Universal Robots PolyScope program: circle motion edge detect.urp

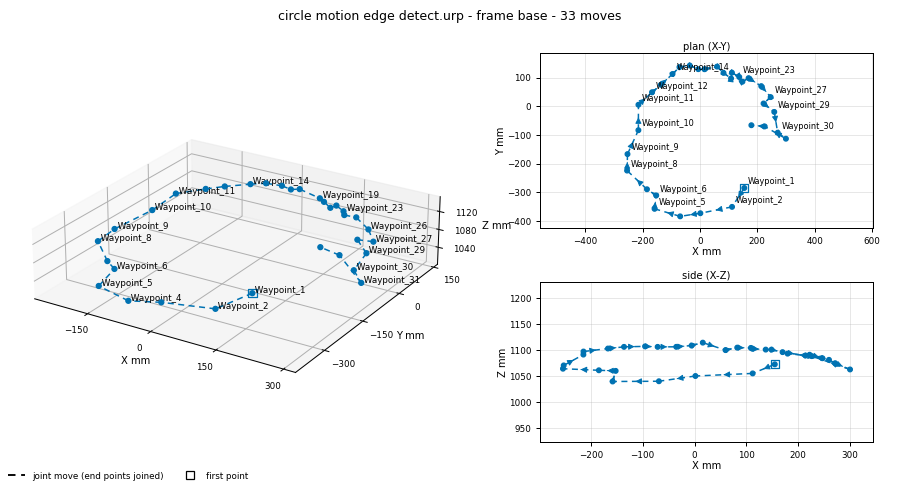
[picture p0: tool path of circle motion edge detect.urp in frame base, 33 of 33 moves have a stored position in this frame; points joined in program order, loops and branches not executed]
Program circle motion edge detect (installation=default directory=/programs/usbdisk createdIn=5.3.0.64176 lastSavedIn=5.3.0.64176 robotSerialNumber=20195500242)
Calibrated DH parameters: a=[-0.00003, -0.418785, -0.364045, -0.000016, 0.000085, 0]; d=[0.162521, -27.105222, -29.89969, 57.138732, 0.099744, 0.099563]; alpha=[1.571361, -0.002704, -0.002569, 1.570134, -1.569255, 0]; deltaTheta=[0, 0.173233, 6.492369, -0.382427, -0.000002, 0]
Robot Program (runOnlyOnce=false)
  MoveJ speed 60 deg/s, acceleration 80 deg/s^2 (useActiveTCP=true) feature=Base
    Waypoint Waypoint_1: TCP in base x=154.914 y=-284.469 z=1072.951 mm, rx=0.2997 ry=-0.5241 rz=-2.3512 rad; joints [-37.372, -111.15, 6.695, -138.52, -90.992, 169.489] deg
    Wait Sleep waitTime=2
    Waypoint Waypoint_2: TCP in base x=112.222 y=-350.291 z=1055.38 mm, rx=0.2716 ry=-0.6364 rz=-2.5729 rad; joints [-51.18, -115.112, 6.722, -132.303, -90.965, 169.471] deg; TCP offset x=0 y=0 z=0 mm, rx=0 ry=0 rz=0 rad
    Wait Sleep waitTime=2
    Waypoint Waypoint_3: TCP in base x=1.771 y=-372.471 z=1050.371 mm, rx=0.1105 ry=-0.864 rz=-2.8765 rad; joints [-70.07, -116.408, 6.715, -126.913, -94.954, 169.472] deg; TCP offset x=0 y=0 z=0 mm, rx=0 ry=0 rz=0 rad
    Wait Sleep waitTime=2
    Waypoint Waypoint_4: TCP in base x=-68.656 y=-383.358 z=1040.258 mm, rx=-0.0416 ry=0.9721 rz=2.9298 rad; joints [-81.366, -118.375, 6.714, -121.793, -94.913, 169.475] deg
    Wait Sleep waitTime=2
    Waypoint Waypoint_5: TCP in base x=-158.009 y=-357.106 z=1039.79 mm, rx=0.0714 ry=0.905 rz=2.7108 rad; joints [-95.142, -118.447, 6.717, -121.809, -94.948, 169.471] deg; TCP offset x=0 y=0 z=0 mm, rx=0 ry=0 rz=0 rad
    Wait Sleep waitTime=2
    Waypoint Waypoint_6: TCP in base x=-152.118 y=-310.493 z=1060.277 mm, rx=0.1283 ry=0.8737 rz=2.7 rad; joints [-95.524, -114.683, 6.715, -126.752, -97.143, 169.442] deg
    Wait Sleep waitTime=2
    Waypoint Waypoint_7: TCP in base x=-184.474 y=-288.892 z=1061.417 mm, rx=0.1713 ry=0.8461 rz=2.5969 rad; joints [-101.799, -114.48, 6.716, -126.753, -97.157, 169.441] deg
    Wait Sleep waitTime=2
    Waypoint Waypoint_8: TCP in base x=-253.787 y=-223.74 z=1064.438 mm, rx=0.2688 ry=0.6858 rz=2.3492 rad; joints [-117.741, -113.528, 6.714, -131.132, -97.725, 169.066] deg
    Wait Sleep waitTime=2
    Waypoint Waypoint_9: TCP in base x=-252.359 y=-166.285 z=1070.795 mm, rx=0.4935 ry=0.5953 rz=1.8556 rad; joints [-127.845, -111.078, 6.717, -133.526, -111.538, 154.842] deg
    Wait Sleep waitTime=2
    Waypoint Waypoint_10: TCP in base x=-214.374 y=-83.001 z=1091.69 mm, rx=0.5264 ry=0.6522 rz=1.7224 rad; joints [-133.832, -106.245, 6.744, -133.513, -111.607, 154.823] deg
    Wait Sleep waitTime=2
    Waypoint Waypoint_11: TCP in base x=-214.184 y=5.835 z=1097.569 mm, rx=0.5409 ry=0.5799 rz=1.432 rad; joints [-152.715, -105.043, 6.723, -133.525, -107.815, 154.808] deg
    Wait Sleep waitTime=2
    Waypoint Waypoint_12: TCP in base x=-166.957 y=49.058 z=1103.38 mm, rx=0.5833 ry=0.3942 rz=1.2936 rad; joints [-161.963, -100.794, 6.708, -143.941, -110.807, 154.793] deg
    Wait Sleep waitTime=2
    Waypoint Waypoint_13: TCP in base x=-136 y=75.302 z=1106.619 mm, rx=0.5655 ry=0.4183 rz=0.9843 rad; joints [-169.727, -99.399, 6.733, -143.942, -110.805, 144.497] deg
    Wait Sleep waitTime=2
    Waypoint Waypoint_14: TCP in base x=-95.348 y=112.97 z=1107.58 mm, rx=0.7237 ry=0.4441 rz=0.5929 rad; joints [-189.526, -100.482, 6.716, -132.699, -112.568, 144.513] deg
    Wait Sleep waitTime=2
    Waypoint Waypoint_15: TCP in base x=-71.129 y=136.814 z=1106.589 mm, rx=0.7608 ry=0.3382 rz=0.3554 rad; joints [-204.168, -100.977, 6.716, -132.715, -112.525, 144.514] deg; TCP offset x=0 y=0 z=0 mm, rx=0 ry=0 rz=0 rad
    Wait Sleep waitTime=2
    Waypoint Waypoint_16: TCP in base x=-35.171 y=142.592 z=1106.68 mm, rx=0.6766 ry=0.1374 rz=0.2072 rad; joints [-215.551, -98.736, 6.732, -144.572, -112.524, 144.514] deg; TCP offset x=0 y=0 z=0 mm, rx=0 ry=0 rz=0 rad
    Wait Sleep waitTime=2
    Waypoint Waypoint_17: TCP in base x=-5.632 y=129.883 z=1109.151 mm, rx=0.6981 ry=0.1269 rz=0.1239 rad; joints [-220.201, -97.319, 6.732, -144.572, -112.523, 144.518] deg; TCP offset x=0 y=0 z=0 mm, rx=0 ry=0 rz=0 rad
    Wait Sleep waitTime=2
    Waypoint Waypoint_18: TCP in base x=15.993 y=129.668 z=1114.734 mm, rx=0.6763 ry=0.2381 rz=0.2822 rad; joints [-220.316, -97.009, 6.71, -140.826, -104.269, 152.017] deg; TCP offset x=0 y=0 z=0 mm, rx=0 ry=0 rz=0 rad
    Wait Sleep waitTime=2
    Waypoint Waypoint_19: TCP in base x=59.885 y=138.766 z=1100.329 mm, rx=0.6524 ry=-0.0476 rz=0.1475 rad; joints [-246.927, -85.881, -20.149, -128.724, -103.816, 169.846] deg; TCP offset x=0 y=0 z=0 mm, rx=0 ry=0 rz=0 rad
    Wait Sleep waitTime=2
    Waypoint Waypoint_20: TCP in base x=82.45 y=116.928 z=1105.125 mm, rx=0.6534 ry=0.2343 rz=-0.2354 rad; joints [-246.975, -84.634, -20.096, -125.99, -96.737, 145.064] deg; TCP offset x=0 y=0 z=0 mm, rx=0 ry=0 rz=0 rad
    Wait Sleep waitTime=2
    Waypoint Waypoint_21: TCP in base x=108.815 y=97.49 z=1104.594 mm, rx=0.6598 ry=0.1537 rz=-0.5229 rad; joints [-261.813, -84.817, -20.066, -127.18, -96.744, 142.73] deg; TCP offset x=0 y=0 z=0 mm, rx=0 ry=0 rz=0 rad
    Wait Sleep waitTime=2
    Waypoint Waypoint_22: TCP in base x=111.731 y=117.75 z=1102.96 mm, rx=0.6639 ry=0.218 rz=-0.5839 rad; joints [-262.695, -86.632, -20.04, -123.996, -94.334, 139.125] deg
    Wait Sleep waitTime=2
    Waypoint Waypoint_23: TCP in base x=137.4 y=102.53 z=1101.341 mm, rx=0.7665 ry=0.2773 rz=-0.7011 rad; joints [-271.96, -88.103, -20.048, -116.073, -89.774, 139.116] deg
    Wait Sleep waitTime=2
    Waypoint Waypoint_24: TCP in base x=148.462 y=86.299 z=1101.282 mm, rx=0.7869 ry=0.2329 rz=-0.8115 rad; joints [-278.669, -88.134, -20.048, -116.076, -89.805, 139.131] deg; TCP offset x=0 y=0 z=0 mm, rx=0 ry=0 rz=0 rad
    Wait Sleep waitTime=2
    Waypoint Waypoint_25: TCP in base x=169.873 y=98.607 z=1096.434 mm, rx=0.7711 ry=0.1697 rz=-0.9529 rad; joints [-286.936, -90.344, -20.046, -116.082, -89.79, 139.118] deg; TCP offset x=0 y=0 z=0 mm, rx=0 ry=0 rz=0 rad
    Wait Sleep waitTime=2
    Waypoint Waypoint_26: TCP in base x=214.106 y=70.755 z=1089.842 mm, rx=0.7695 ry=0.0439 rz=-1.2633 rad; joints [-305.319, -92.663, -20.048, -116.082, -89.78, 139.118] deg
    Wait Sleep waitTime=2
    Waypoint Waypoint_27: TCP in base x=246.914 y=32.42 z=1084.615 mm, rx=0.7637 ry=0.0266 rz=-1.459 rad; joints [-318.237, -94.154, -20.051, -116.079, -86.045, 139.124] deg; TCP offset x=0 y=0 z=0 mm, rx=0 ry=0 rz=0 rad
    Wait Sleep waitTime=2
    Waypoint Waypoint_28: TCP in base x=222.111 y=10.22 z=1091.429 mm, rx=0.7745 ry=-0.0817 rz=-1.1956 rad; joints [-318.239, -92.102, -20.038, -116.074, -86.03, 154.561] deg
    Wait Sleep waitTime=2
    Waypoint Waypoint_29: TCP in base x=259.462 y=-19.167 z=1081.558 mm, rx=0.7346 ry=-0.1451 rz=-1.4632 rad; joints [-331.589, -94.992, -20.034, -116.079, -86.026, 152.414] deg
    Wait Sleep waitTime=2
    Waypoint Waypoint_30: TCP in base x=271.355 y=-91.552 z=1075.114 mm, rx=0.5548 ry=-0.2647 rz=-1.4958 rad; joints [-349.009, -95.902, -20.026, -122.396, -85.227, 169.208] deg; TCP offset x=0 y=0 z=0 mm, rx=0 ry=0 rz=0 rad
    Wait Sleep waitTime=2
    Waypoint Waypoint_31: TCP in base x=300.078 y=-112.654 z=1063.014 mm, rx=0.587 ry=-0.2983 rz=-1.5634 rad; joints [-353.999, -99.028, -20.028, -117.453, -84.219, 169.468] deg; TCP offset x=0 y=0 z=0 mm, rx=0 ry=0 rz=0 rad
    Wait Sleep waitTime=2
    Waypoint Waypoint_32: TCP in base x=226.129 y=-69.813 z=1088.712 mm, rx=0.4806 ry=-0.2241 rz=-1.1145 rad; joints [-339.929, -90.898, -20.032, -130.72, -84.265, 182.917] deg
    Wait Sleep waitTime=2
    Waypoint Waypoint_33: TCP in base x=179.612 y=-65.598 z=1093.539 mm, rx=0.4063 ry=-0.0783 rz=-1.165 rad; joints [-331.319, -85.3, -20.048, -143.011, -83.853, 172.223] deg; TCP offset x=0 y=0 z=0 mm, rx=0 ry=0 rz=0 rad
